# EPICS autosave request: laudaRE2xx/lRE2xx_RS485_settings.req
$(P):DISABLE
$(P):SET_TEMP
